INTERFACE iUPS

(*
Method of saving persistent data
=================================================

Author
	: Takashi Ichihashi

Date
	: 02 Aug, 2023

Overview
===============

This method is assumed that persistent values are saved when ups running without online power.
"WritePersistentData" FB has to be executed explicily in case of GenericUPS is used. You might define this FB instance on this method.
If you use "SUPS", it might be saved persistent data automatically when power failed, so nothing need to be defined on this method.

*)
METHOD persist_data : BOOL
VAR_INPUT
END_VAR
END_METHOD

METHOD shutdown : BOOL
VAR_INPUT
END_VAR
END_METHOD

PROPERTY shutdown_delay : TIME
GET
END_GET
SET
END_SET
END_PROPERTY

PROPERTY UPSState : E_UPSState
GET
END_GET
END_PROPERTY

METHOD watch_status : BOOL
VAR_INPUT
END_VAR
END_METHOD

END_INTERFACE

(* stored: Version 1.1.0.1, ProductVersion 3.1.4024.12
   Itf iUPS: Id {a3d4dadb-cbcc-45dc-9c32-777e8f010ae0}
   Method persist_data: Id {75e31577-948a-4c0e-a956-0acb791fdeba}
   Method shutdown: Id {cc96a78c-d834-4b2b-a85b-51732d332b57}
   Property shutdown_delay: Id {b6287d37-5af7-4592-877d-72d17bf7b41a}
   Get Get: Id {90f23270-b879-4949-a87f-752d7c423c5c}
   Set Set: Id {7aa59039-fd9e-4e53-896c-55dc2e9b5c8b}
   Property UPSState: Id {b3b83b4b-f94c-4f6a-a48c-b02264ac592a}
   Get Get: Id {0300f15b-e905-49b7-a86b-afff88d77d7c}
   Method watch_status: Id {636be49c-911a-4fbc-aece-b7a3c5ae21c9} *)
